(* Logix 5000 project; controller PLC vendor 1 type 14 code 155 rev 32.13; software revision 32.04; part 3 of 5 *)
(* tags used below, declared in another part *)
   Alarm_Word_Current : DINT[3];
   Bridge_Timer_Gearing_Delay : TIMER;
   Bridge_Timer_Gearing_Delay_DN_OS : BOOL;
   Bypass_Encoder : BOOL;   // HMI ENABLE ENCODER
   Depositor : Depositor_R2b;
   FORCE_GO_SIGNAL : BOOL;
   Forces : Forces_R2b;
   homing_timeout : TIMER;
   IO : IO_R2a;
   mv_index_counter : COUNTER;
   MV_indexes : DINT;
   MV_total_indexes : COUNTER;
   NC_NF : NCNF_R2a;   // NC/NF BITSHIFTS
   OS : INT[10];
   Recipe_Setpoints_DINT : DINT[23,20];
   Sequencer_Auto : Sequencer_R2a;
   Sequencer_Home : Sequencer_R2a;
   Servo_MC_Bridge_Shift : Axis_MC_R3b;
   System : System_R2e;
   Timer_Done_Signal_Pulse : TIMER;
   Timers : TIMER[20];   // x
(* MainProgram, continued *)

ROUTINE File_012_Digital_Outputs   (* ladder *)
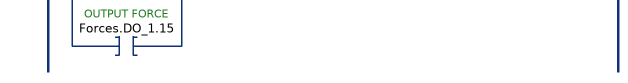
   // DIGITAL OUTPUT MAPPING
   0: [[XIC(IO.DO_1.0) ,XIC(Forces.DO_1.0) ] OTE(Local:1:O.Data.0) ,[XIC(IO.DO_1.1) ,XIC(Forces.DO_1.1) ] OTE(Local:1:O.Data.1) ,[XIC(IO.DO_1.2) ,XIC(Forces.DO_1.2) ] OTE(Local:1:O.Data.2) ,[XIC(IO.DO_1.3) ,XIC(Forces.DO_1.3) ] OTE(Local:1:O.Data.3) ,[XIC(IO.DO_1.4) ,XIC(Forces.DO_1.4) ] OTE(Local:1:O.Data.4) ,[XIC(IO.DO_1.5) ,XIC(Forces.DO_1.5) ] OTE(Local:1:O.Data.5) ,[XIC(IO.DO_1.6) ,XIC(Forces.DO_1.6) ] OTE(Local:1:O.Data.6) ,[XIC(IO.DO_1.7) ,XIC(Forces.DO_1.7) ] OTE(Local:1:O.Data.7) ,[XIC(IO.DO_1.8) ,XIC(Forces.DO_1.8) ] OTE(Local:1:O.Data.8) ,[XIC(IO.DO_1.9) ,XIC(Forces.DO_1.9) ] OTE(Local:1:O.Data.9) ,[XIC(IO.DO_1.10) ,XIC(Forces.DO_1.10) ] OTE(Local:1:O.Data.10) ,[XIC(IO.DO_1.11) ,XIC(Forces.DO_1.11) ] OTE(Local:1:O.Data.11) ,[XIC(IO.DO_1.12) ,XIC(Forces.DO_1.12) ] OTE(Local:1:O.Data.12) ,[XIC(IO.DO_1.13) ,XIC(Forces.DO_1.13) ] OTE(Local:1:O.Data.13) ,[XIC(IO.DO_1.14) ,XIC(Forces.DO_1.14) ] OTE(Local:1:O.Data.14) ,[XIC(IO.DO_1.15) ,XIC(Forces.DO_1.15) ] OTE(Local:1:O.Data.15) ];
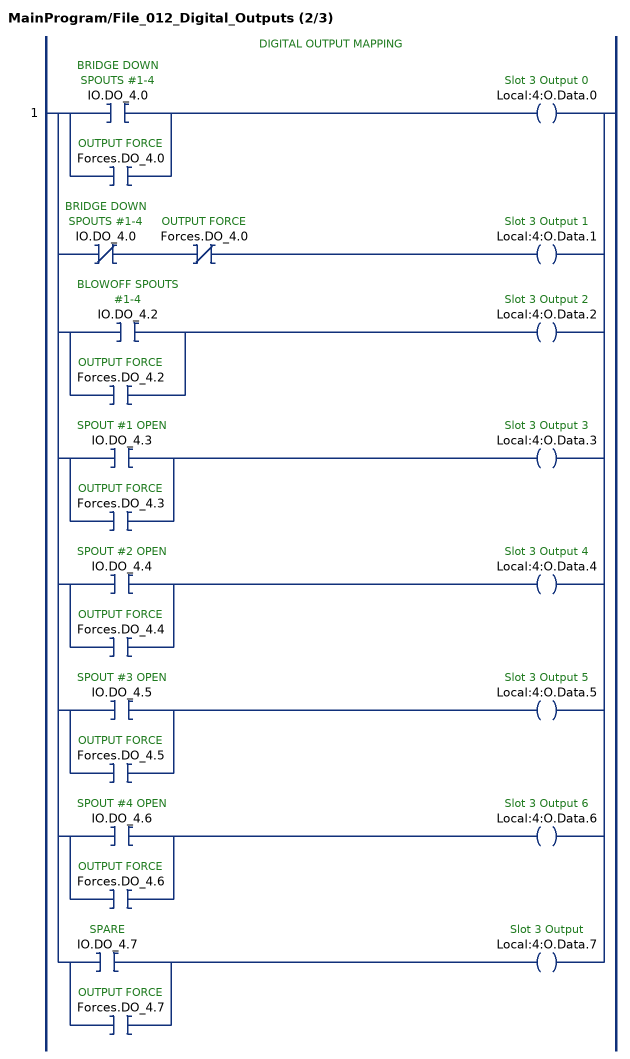
   // DIGITAL OUTPUT MAPPING
   1: [[XIC(IO.DO_4.0) ,XIC(Forces.DO_4.0) ] OTE(Local:4:O.Data.0) ,XIO(IO.DO_4.0) XIO(Forces.DO_4.0) OTE(Local:4:O.Data.1) ,[XIC(IO.DO_4.2) ,XIC(Forces.DO_4.2) ] OTE(Local:4:O.Data.2) ,[XIC(IO.DO_4.3) ,XIC(Forces.DO_4.3) ] OTE(Local:4:O.Data.3) ,[XIC(IO.DO_4.4) ,XIC(Forces.DO_4.4) ] OTE(Local:4:O.Data.4) ,[XIC(IO.DO_4.5) ,XIC(Forces.DO_4.5) ] OTE(Local:4:O.Data.5) ,[XIC(IO.DO_4.6) ,XIC(Forces.DO_4.6) ] OTE(Local:4:O.Data.6) ,[XIC(IO.DO_4.7) ,XIC(Forces.DO_4.7) ] OTE(Local:4:O.Data.7) ];
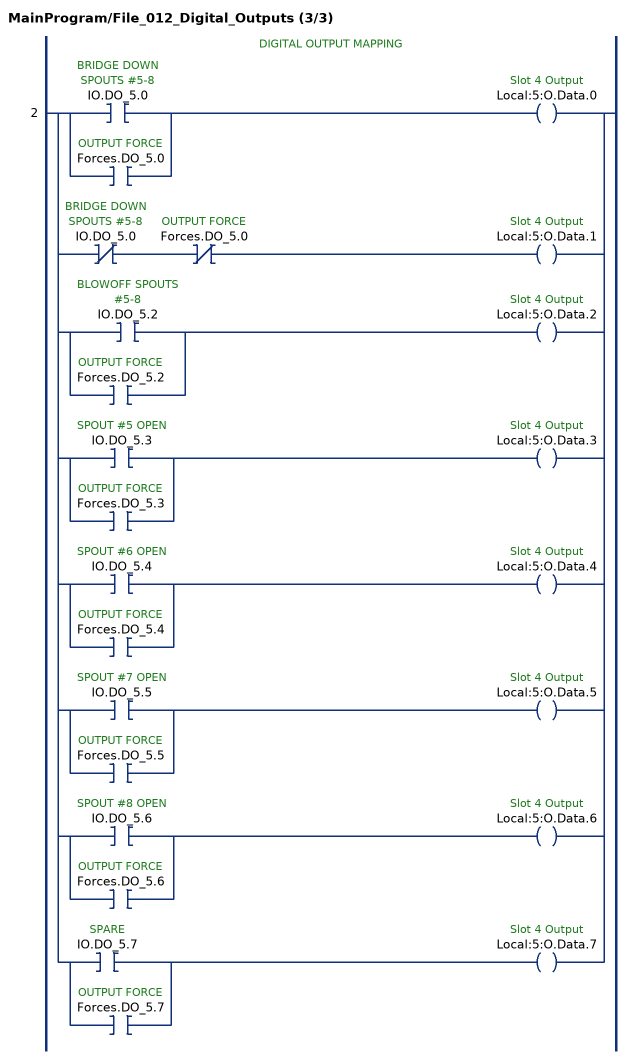
   // DIGITAL OUTPUT MAPPING
   2: [[XIC(IO.DO_5.0) ,XIC(Forces.DO_5.0) ] OTE(Local:5:O.Data.0) ,XIO(IO.DO_5.0) XIO(Forces.DO_5.0) OTE(Local:5:O.Data.1) ,[XIC(IO.DO_5.2) ,XIC(Forces.DO_5.2) ] OTE(Local:5:O.Data.2) ,[XIC(IO.DO_5.3) ,XIC(Forces.DO_5.3) ] OTE(Local:5:O.Data.3) ,[XIC(IO.DO_5.4) ,XIC(Forces.DO_5.4) ] OTE(Local:5:O.Data.4) ,[XIC(IO.DO_5.5) ,XIC(Forces.DO_5.5) ] OTE(Local:5:O.Data.5) ,[XIC(IO.DO_5.6) ,XIC(Forces.DO_5.6) ] OTE(Local:5:O.Data.6) ,[XIC(IO.DO_5.7) ,XIC(Forces.DO_5.7) ] OTE(Local:5:O.Data.7) ];
END_ROUTINE

ROUTINE File_030_Sequencer_Homing   (* ladder *)
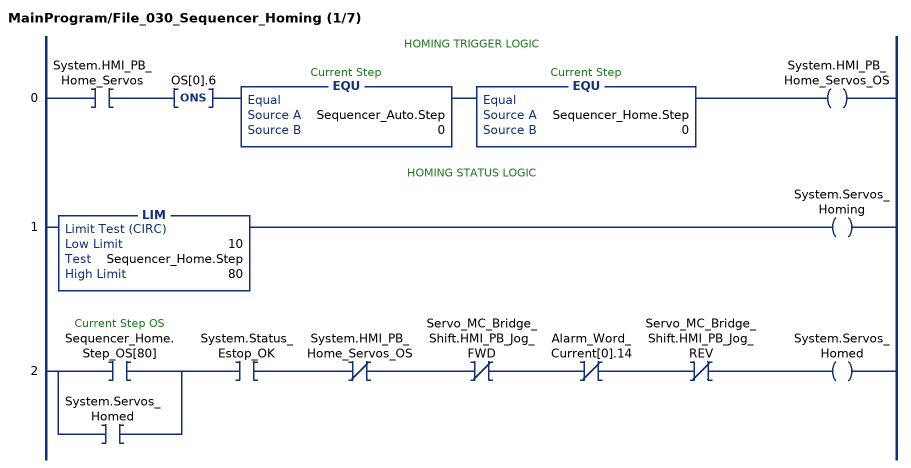
   // HOMING TRIGGER LOGIC
   0: XIC(System.HMI_PB_Home_Servos)ONS(OS[0].6)EQU(Sequencer_Auto.Step,0)EQU(Sequencer_Home.Step,0)OTE(System.HMI_PB_Home_Servos_OS);
   // HOMING STATUS LOGIC
   1: LIM(10,Sequencer_Home.Step,80)OTE(System.Servos_Homing);
   2: [XIC(Sequencer_Home.Step_OS[80]) ,XIC(System.Servos_Homed) ]XIC(System.Status_Estop_OK)XIO(System.HMI_PB_Home_Servos_OS)XIO(Servo_MC_Bridge_Shift.HMI_PB_Jog_FWD)XIO(Alarm_Word_Current[0].14)XIO(Servo_MC_Bridge_Shift.HMI_PB_Jog_REV)OTE(System.Servos_Homed);
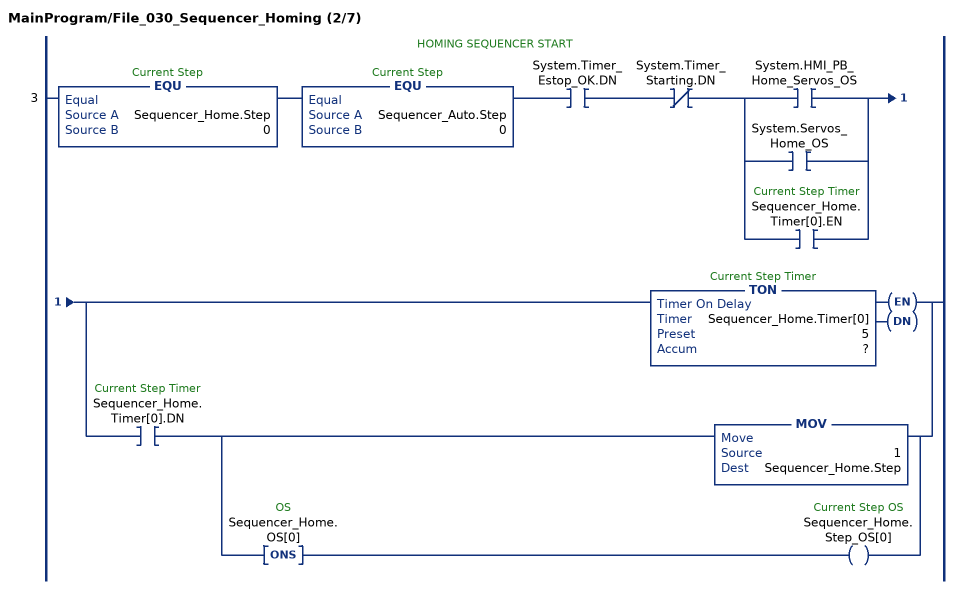
   // HOMING SEQUENCER START
   3: EQU(Sequencer_Home.Step,0)EQU(Sequencer_Auto.Step,0)XIC(System.Timer_Estop_OK.DN)XIO(System.Timer_Starting.DN)[XIC(System.HMI_PB_Home_Servos_OS) ,XIC(System.Servos_Home_OS) ,XIC(Sequencer_Home.Timer[0].EN) ][TON(Sequencer_Home.Timer[0],?,?) ,XIC(Sequencer_Home.Timer[0].DN) [MOV(1,Sequencer_Home.Step) ,ONS(Sequencer_Home.OS[0]) OTE(Sequencer_Home.Step_OS[0]) ] ];
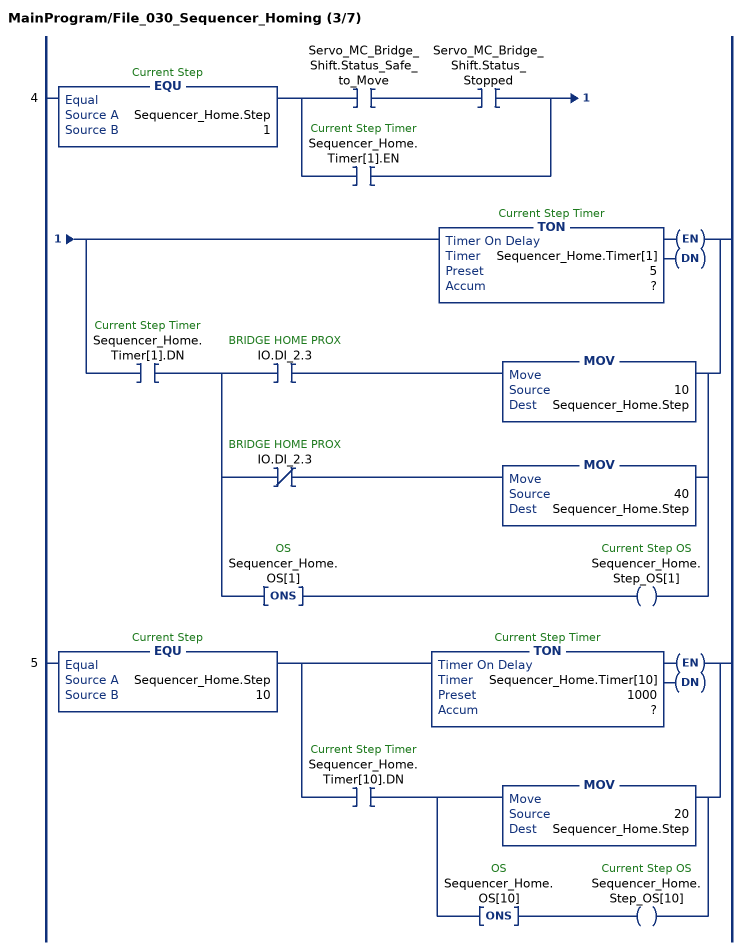
   4: EQU(Sequencer_Home.Step,1)[XIC(Servo_MC_Bridge_Shift.Status_Safe_to_Move) XIC(Servo_MC_Bridge_Shift.Status_Stopped) ,XIC(Sequencer_Home.Timer[1].EN) ][TON(Sequencer_Home.Timer[1],?,?) ,XIC(Sequencer_Home.Timer[1].DN) [XIC(IO.DI_2.3) MOV(10,Sequencer_Home.Step) ,XIO(IO.DI_2.3) MOV(40,Sequencer_Home.Step) ,ONS(Sequencer_Home.OS[1]) OTE(Sequencer_Home.Step_OS[1]) ] ];
   5: EQU(Sequencer_Home.Step,10)[TON(Sequencer_Home.Timer[10],?,?) ,XIC(Sequencer_Home.Timer[10].DN) [MOV(20,Sequencer_Home.Step) ,ONS(Sequencer_Home.OS[10]) OTE(Sequencer_Home.Step_OS[10]) ] ];
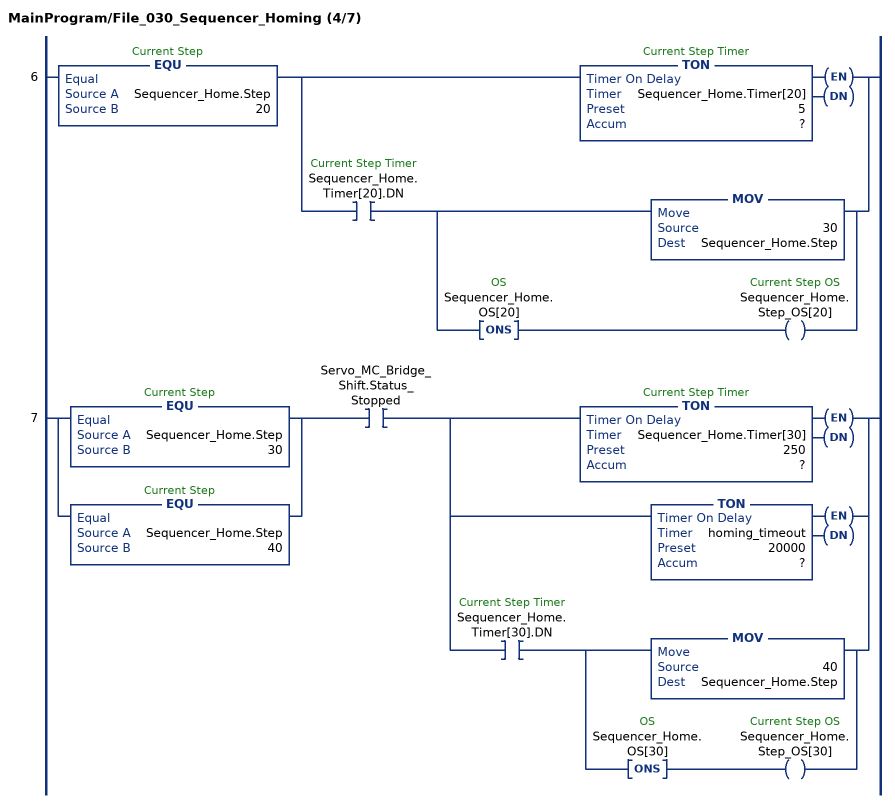
   6: EQU(Sequencer_Home.Step,20)[TON(Sequencer_Home.Timer[20],?,?) ,XIC(Sequencer_Home.Timer[20].DN) [MOV(30,Sequencer_Home.Step) ,ONS(Sequencer_Home.OS[20]) OTE(Sequencer_Home.Step_OS[20]) ] ];
   7: [EQU(Sequencer_Home.Step,30) ,EQU(Sequencer_Home.Step,40) ]XIC(Servo_MC_Bridge_Shift.Status_Stopped)[[TON(Sequencer_Home.Timer[30],?,?) ,TON(homing_timeout,?,?) ] ,XIC(Sequencer_Home.Timer[30].DN) [MOV(40,Sequencer_Home.Step) ,ONS(Sequencer_Home.OS[30]) OTE(Sequencer_Home.Step_OS[30]) ] ];
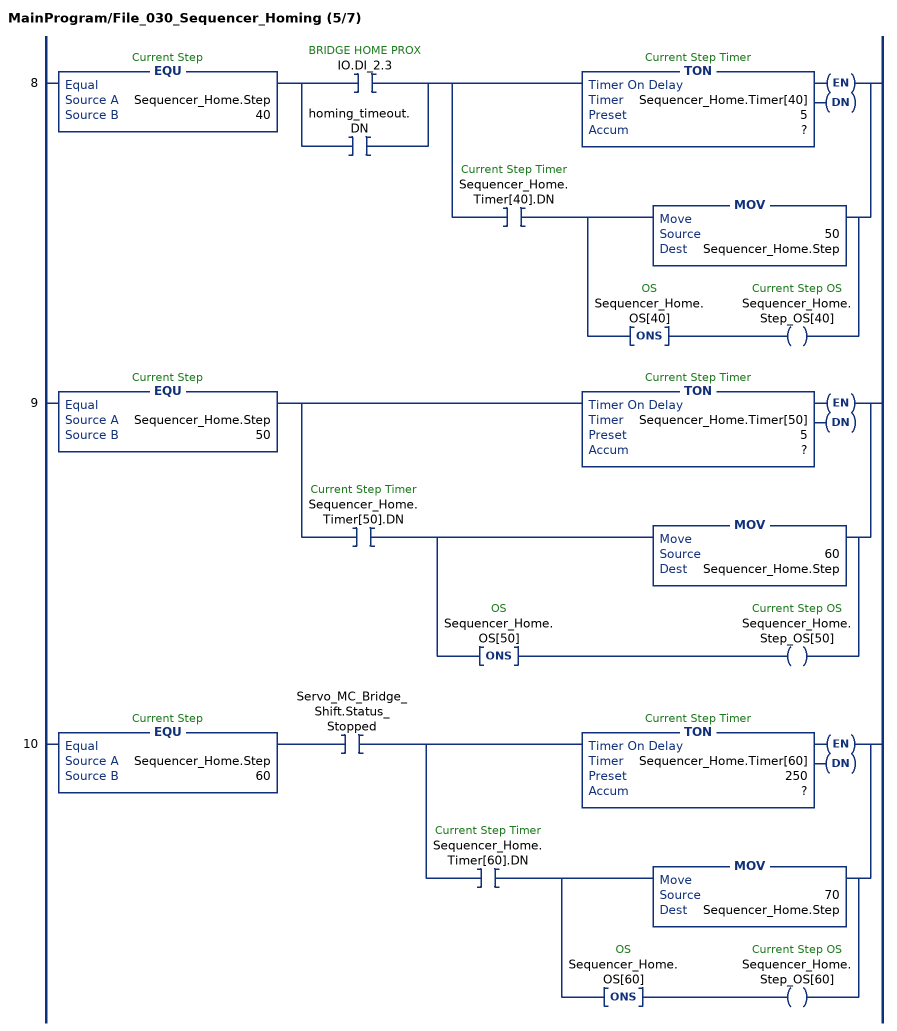
   8: EQU(Sequencer_Home.Step,40)[XIC(IO.DI_2.3) ,XIC(homing_timeout.DN) ][TON(Sequencer_Home.Timer[40],?,?) ,XIC(Sequencer_Home.Timer[40].DN) [MOV(50,Sequencer_Home.Step) ,ONS(Sequencer_Home.OS[40]) OTE(Sequencer_Home.Step_OS[40]) ] ];
   9: EQU(Sequencer_Home.Step,50)[TON(Sequencer_Home.Timer[50],?,?) ,XIC(Sequencer_Home.Timer[50].DN) [MOV(60,Sequencer_Home.Step) ,ONS(Sequencer_Home.OS[50]) OTE(Sequencer_Home.Step_OS[50]) ] ];
   10: EQU(Sequencer_Home.Step,60)XIC(Servo_MC_Bridge_Shift.Status_Stopped)[TON(Sequencer_Home.Timer[60],?,?) ,XIC(Sequencer_Home.Timer[60].DN) [MOV(70,Sequencer_Home.Step) ,ONS(Sequencer_Home.OS[60]) OTE(Sequencer_Home.Step_OS[60]) ] ];
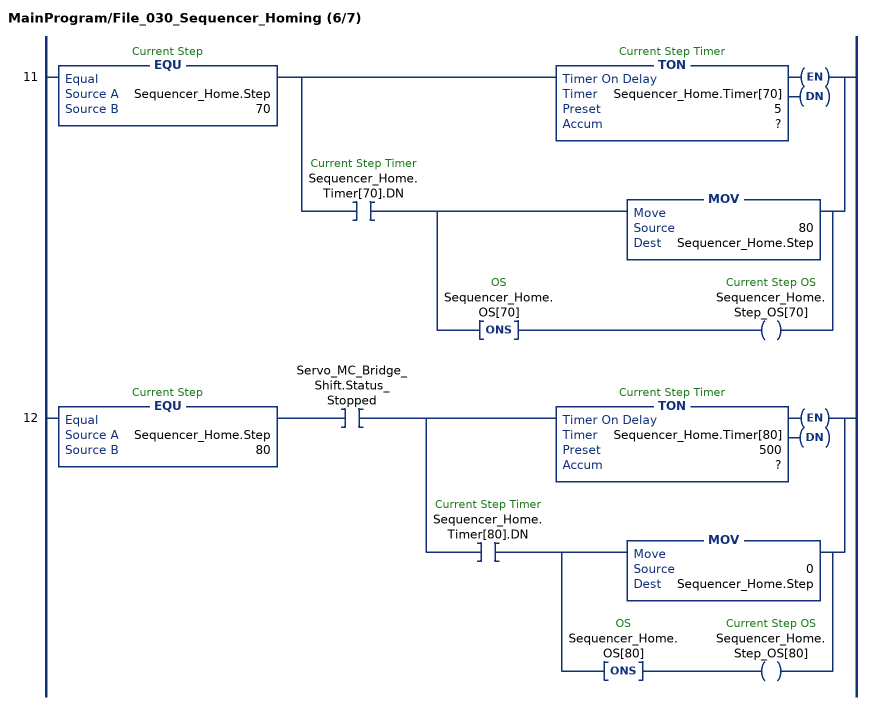
   11: EQU(Sequencer_Home.Step,70)[TON(Sequencer_Home.Timer[70],?,?) ,XIC(Sequencer_Home.Timer[70].DN) [MOV(80,Sequencer_Home.Step) ,ONS(Sequencer_Home.OS[70]) OTE(Sequencer_Home.Step_OS[70]) ] ];
   12: EQU(Sequencer_Home.Step,80)XIC(Servo_MC_Bridge_Shift.Status_Stopped)[TON(Sequencer_Home.Timer[80],?,?) ,XIC(Sequencer_Home.Timer[80].DN) [MOV(0,Sequencer_Home.Step) ,ONS(Sequencer_Home.OS[80]) OTE(Sequencer_Home.Step_OS[80]) ] ];
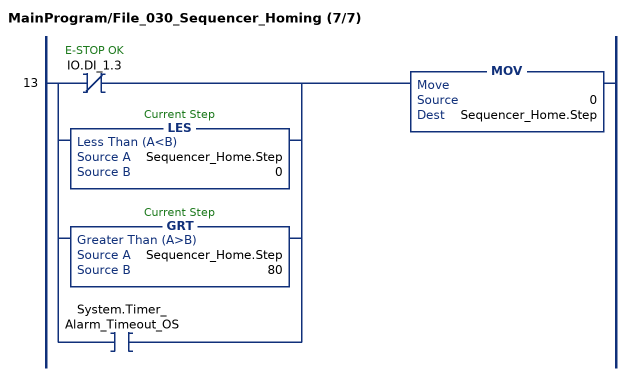
   13: [XIO(IO.DI_1.3) ,LES(Sequencer_Home.Step,0) ,GRT(Sequencer_Home.Step,80) ,XIC(System.Timer_Alarm_Timeout_OS) ]MOV(0,Sequencer_Home.Step);
END_ROUTINE

ROUTINE File_040_Sequencer_Auto   (* ladder *)
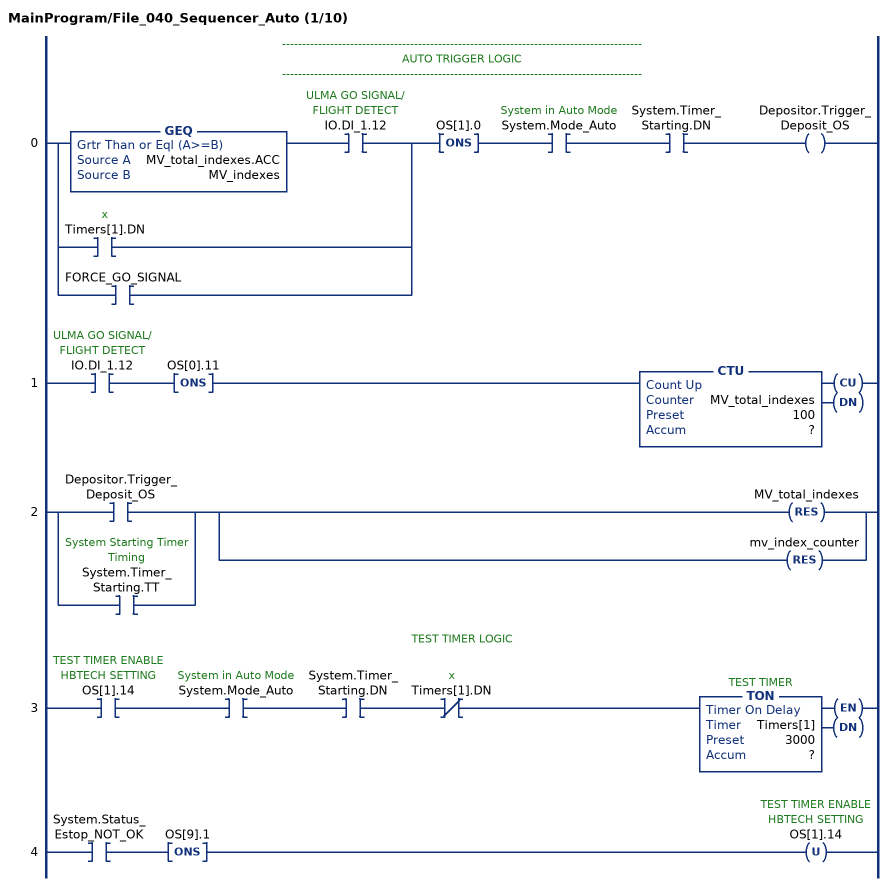
   // ------------------------------------------------------------------------------------------
   // AUTO TRIGGER LOGIC
   // ------------------------------------------------------------------------------------------
   0: [GEQ(MV_total_indexes.ACC,MV_indexes) XIC(IO.DI_1.12) ,XIC(Timers[1].DN) ,XIC(FORCE_GO_SIGNAL) ]ONS(OS[1].0)XIC(System.Mode_Auto)XIC(System.Timer_Starting.DN)OTE(Depositor.Trigger_Deposit_OS);
   1: XIC(IO.DI_1.12)ONS(OS[0].11)CTU(MV_total_indexes,?,?);
   2: [XIC(Depositor.Trigger_Deposit_OS) ,XIC(System.Timer_Starting.TT) ][RES(MV_total_indexes) ,RES(mv_index_counter) ];
   // TEST TIMER LOGIC
   3: XIC(OS[1].14)XIC(System.Mode_Auto)XIC(System.Timer_Starting.DN)XIO(Timers[1].DN)TON(Timers[1],?,?);
   4: XIC(System.Status_Estop_NOT_OK)ONS(OS[9].1)OTU(OS[1].14);
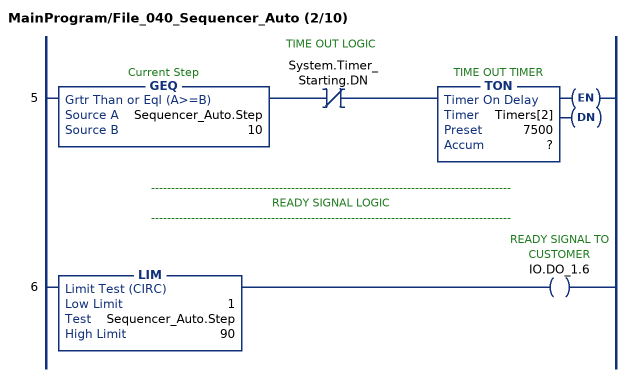
   // TIME OUT LOGIC
   5: GEQ(Sequencer_Auto.Step,10)XIO(System.Timer_Starting.DN)TON(Timers[2],?,?);
   // ------------------------------------------------------------------------------------------
   // READY SIGNAL LOGIC
   // ------------------------------------------------------------------------------------------
   6: LIM(1,Sequencer_Auto.Step,90)OTE(IO.DO_1.6);
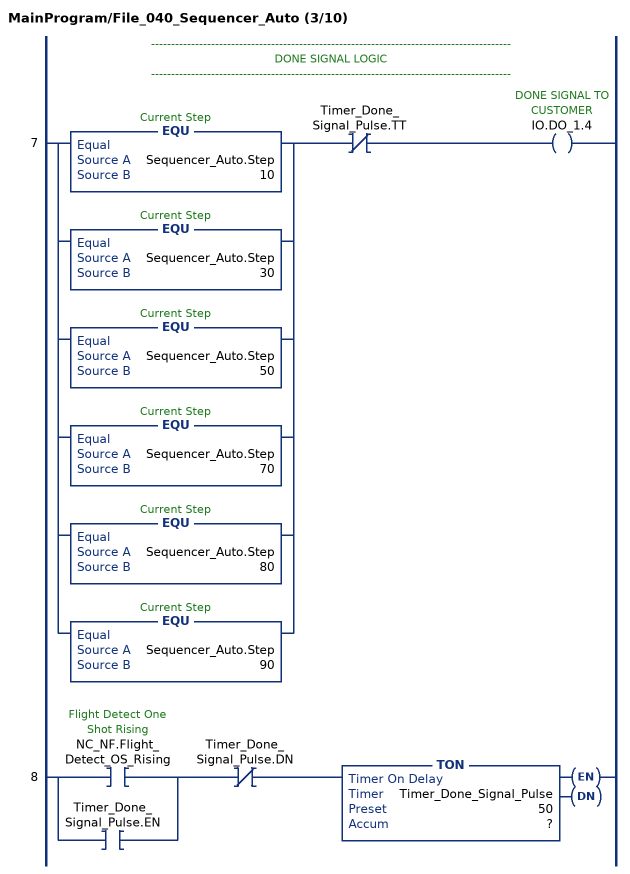
   // ------------------------------------------------------------------------------------------
   // DONE SIGNAL LOGIC
   // ------------------------------------------------------------------------------------------
   7: [EQU(Sequencer_Auto.Step,10) ,EQU(Sequencer_Auto.Step,30) ,EQU(Sequencer_Auto.Step,50) ,EQU(Sequencer_Auto.Step,70) ,EQU(Sequencer_Auto.Step,80) ,EQU(Sequencer_Auto.Step,90) ]XIO(Timer_Done_Signal_Pulse.TT)OTE(IO.DO_1.4);
   8: [XIC(NC_NF.Flight_Detect_OS_Rising) ,XIC(Timer_Done_Signal_Pulse.EN) ]XIO(Timer_Done_Signal_Pulse.DN)TON(Timer_Done_Signal_Pulse,?,?);
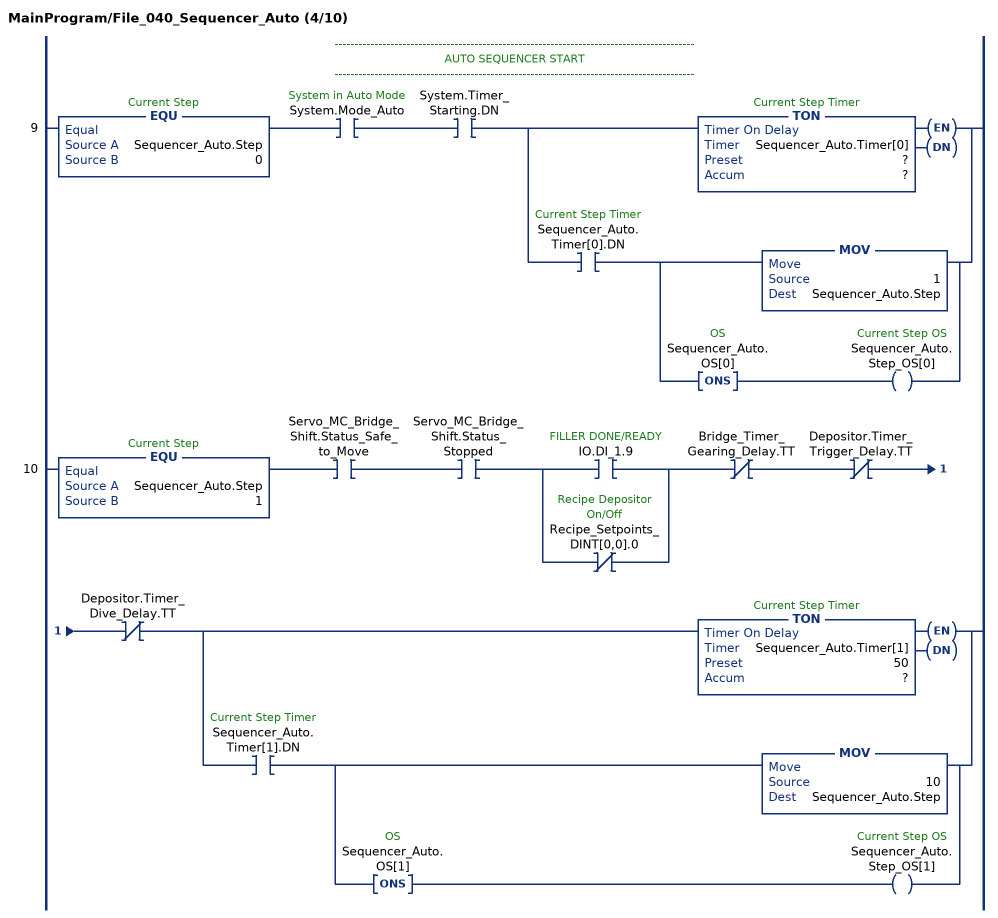
   // ------------------------------------------------------------------------------------------
   // AUTO SEQUENCER START
   // ------------------------------------------------------------------------------------------
   9: EQU(Sequencer_Auto.Step,0)XIC(System.Mode_Auto)XIC(System.Timer_Starting.DN)[TON(Sequencer_Auto.Timer[0],?,?) ,XIC(Sequencer_Auto.Timer[0].DN) [MOV(1,Sequencer_Auto.Step) ,ONS(Sequencer_Auto.OS[0]) OTE(Sequencer_Auto.Step_OS[0]) ] ];
   10: EQU(Sequencer_Auto.Step,1)XIC(Servo_MC_Bridge_Shift.Status_Safe_to_Move)XIC(Servo_MC_Bridge_Shift.Status_Stopped)[XIC(IO.DI_1.9) ,XIO(Recipe_Setpoints_DINT[0,0].0) ]XIO(Bridge_Timer_Gearing_Delay.TT)XIO(Depositor.Timer_Trigger_Delay.TT)XIO(Depositor.Timer_Dive_Delay.TT)[TON(Sequencer_Auto.Timer[1],?,?) ,XIC(Sequencer_Auto.Timer[1].DN) [MOV(10,Sequencer_Auto.Step) ,ONS(Sequencer_Auto.OS[1]) OTE(Sequencer_Auto.Step_OS[1]) ] ];
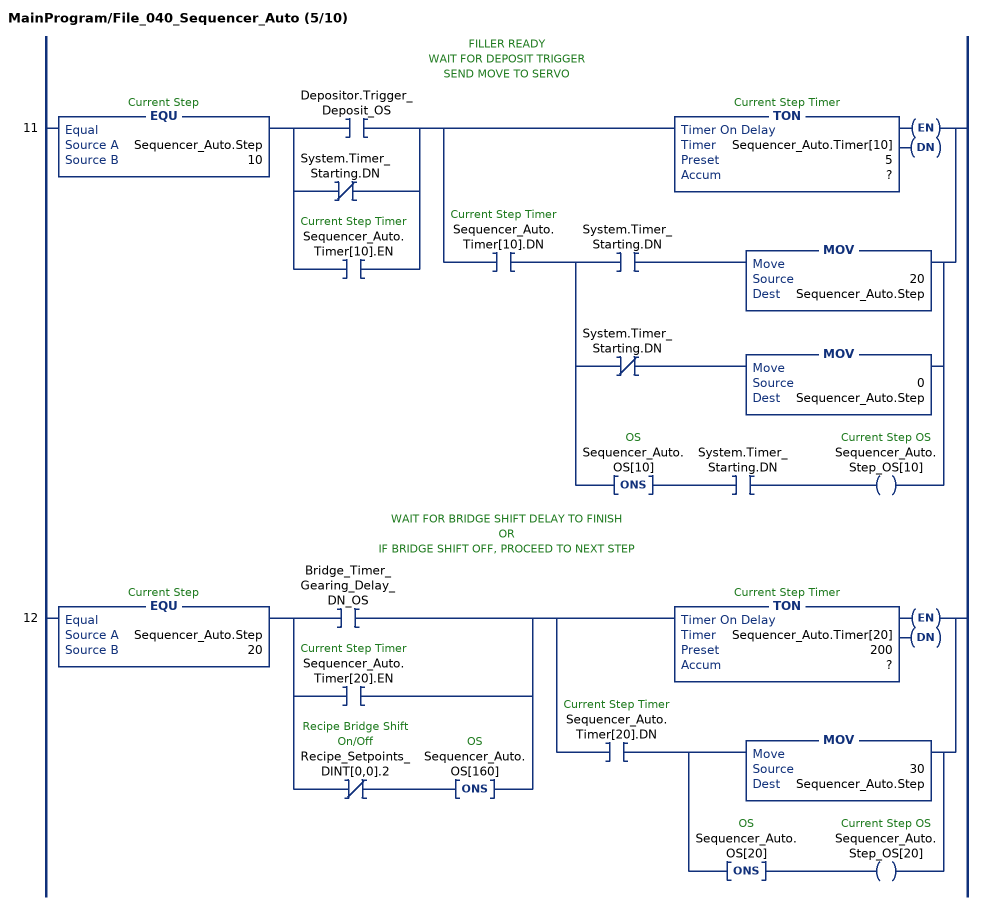
   // FILLER READY
   // WAIT FOR DEPOSIT TRIGGER
   // SEND MOVE TO SERVO
   11: EQU(Sequencer_Auto.Step,10)[XIC(Depositor.Trigger_Deposit_OS) ,XIO(System.Timer_Starting.DN) ,XIC(Sequencer_Auto.Timer[10].EN) ][TON(Sequencer_Auto.Timer[10],?,?) ,XIC(Sequencer_Auto.Timer[10].DN) [XIC(System.Timer_Starting.DN) MOV(20,Sequencer_Auto.Step) ,XIO(System.Timer_Starting.DN) MOV(0,Sequencer_Auto.Step) ,ONS(Sequencer_Auto.OS[10]) XIC(System.Timer_Starting.DN) OTE(Sequencer_Auto.Step_OS[10]) ] ];
   // WAIT FOR BRIDGE SHIFT DELAY TO FINISH
   // OR
   // IF BRIDGE SHIFT OFF, PROCEED TO NEXT STEP
   12: EQU(Sequencer_Auto.Step,20)[XIC(Bridge_Timer_Gearing_Delay_DN_OS) ,XIC(Sequencer_Auto.Timer[20].EN) ,XIO(Recipe_Setpoints_DINT[0,0].2) ONS(Sequencer_Auto.OS[160]) ][TON(Sequencer_Auto.Timer[20],?,?) ,XIC(Sequencer_Auto.Timer[20].DN) [MOV(30,Sequencer_Auto.Step) ,ONS(Sequencer_Auto.OS[20]) OTE(Sequencer_Auto.Step_OS[20]) ] ];
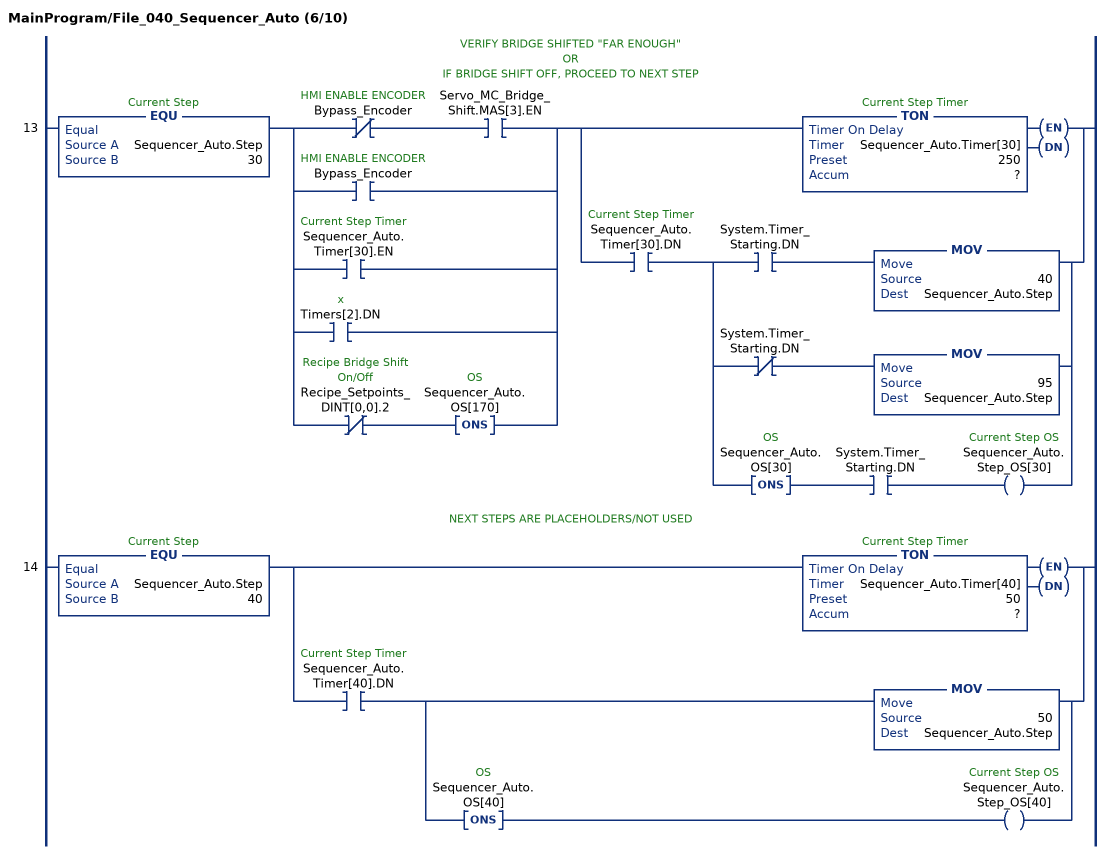
   // VERIFY BRIDGE SHIFTED "FAR ENOUGH"
   // OR
   // IF BRIDGE SHIFT OFF, PROCEED TO NEXT STEP
   13: EQU(Sequencer_Auto.Step,30)[XIO(Bypass_Encoder) XIC(Servo_MC_Bridge_Shift.MAS[3].EN) ,XIC(Bypass_Encoder) ,XIC(Sequencer_Auto.Timer[30].EN) ,XIC(Timers[2].DN) ,XIO(Recipe_Setpoints_DINT[0,0].2) ONS(Sequencer_Auto.OS[170]) ][TON(Sequencer_Auto.Timer[30],?,?) ,XIC(Sequencer_Auto.Timer[30].DN) [XIC(System.Timer_Starting.DN) MOV(40,Sequencer_Auto.Step) ,XIO(System.Timer_Starting.DN) MOV(95,Sequencer_Auto.Step) ,ONS(Sequencer_Auto.OS[30]) XIC(System.Timer_Starting.DN) OTE(Sequencer_Auto.Step_OS[30]) ] ];
   // NEXT STEPS ARE PLACEHOLDERS/NOT USED
   14: EQU(Sequencer_Auto.Step,40)[TON(Sequencer_Auto.Timer[40],?,?) ,XIC(Sequencer_Auto.Timer[40].DN) [MOV(50,Sequencer_Auto.Step) ,ONS(Sequencer_Auto.OS[40]) OTE(Sequencer_Auto.Step_OS[40]) ] ];
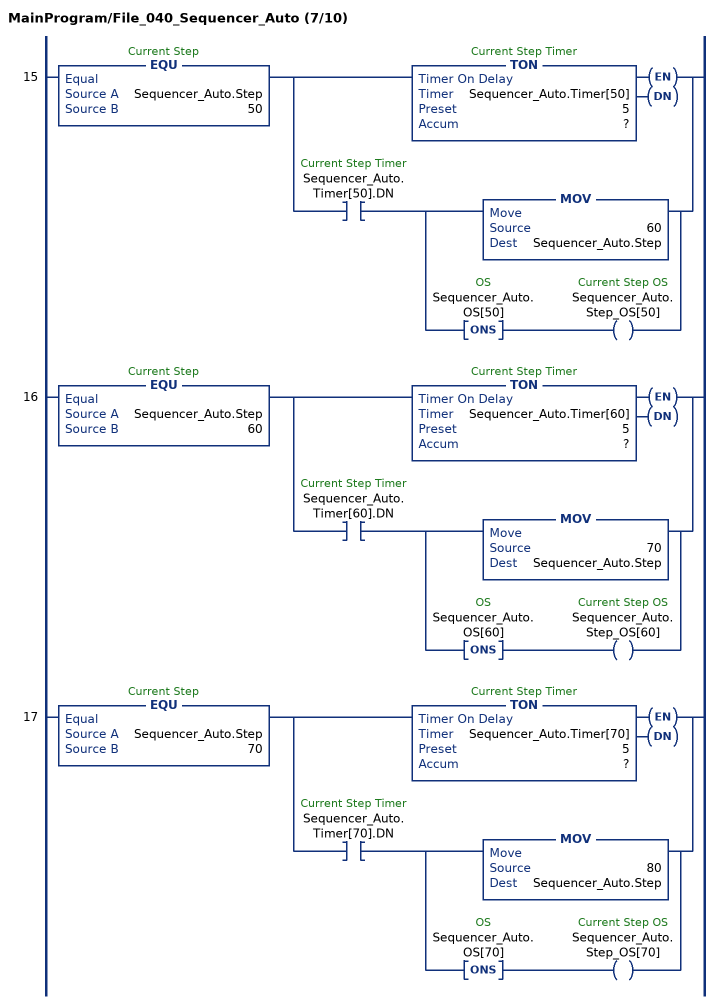
   15: EQU(Sequencer_Auto.Step,50)[TON(Sequencer_Auto.Timer[50],?,?) ,XIC(Sequencer_Auto.Timer[50].DN) [MOV(60,Sequencer_Auto.Step) ,ONS(Sequencer_Auto.OS[50]) OTE(Sequencer_Auto.Step_OS[50]) ] ];
   16: EQU(Sequencer_Auto.Step,60)[TON(Sequencer_Auto.Timer[60],?,?) ,XIC(Sequencer_Auto.Timer[60].DN) [MOV(70,Sequencer_Auto.Step) ,ONS(Sequencer_Auto.OS[60]) OTE(Sequencer_Auto.Step_OS[60]) ] ];
   17: EQU(Sequencer_Auto.Step,70)[TON(Sequencer_Auto.Timer[70],?,?) ,XIC(Sequencer_Auto.Timer[70].DN) [MOV(80,Sequencer_Auto.Step) ,ONS(Sequencer_Auto.OS[70]) OTE(Sequencer_Auto.Step_OS[70]) ] ];
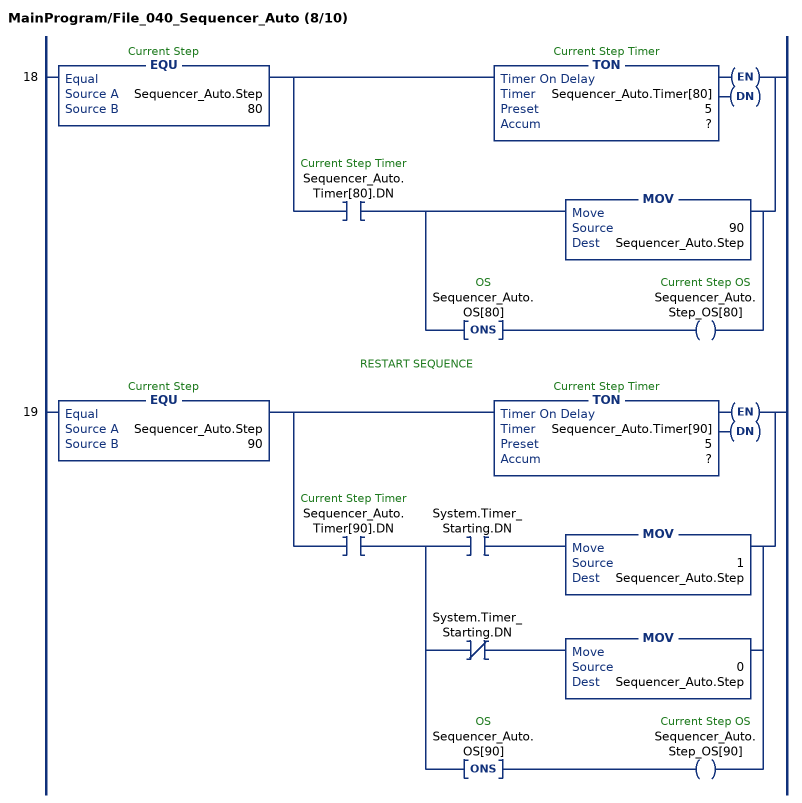
   18: EQU(Sequencer_Auto.Step,80)[TON(Sequencer_Auto.Timer[80],?,?) ,XIC(Sequencer_Auto.Timer[80].DN) [MOV(90,Sequencer_Auto.Step) ,ONS(Sequencer_Auto.OS[80]) OTE(Sequencer_Auto.Step_OS[80]) ] ];
   // RESTART SEQUENCE
   19: EQU(Sequencer_Auto.Step,90)[TON(Sequencer_Auto.Timer[90],?,?) ,XIC(Sequencer_Auto.Timer[90].DN) [XIC(System.Timer_Starting.DN) MOV(1,Sequencer_Auto.Step) ,XIO(System.Timer_Starting.DN) MOV(0,Sequencer_Auto.Step) ,ONS(Sequencer_Auto.OS[90]) OTE(Sequencer_Auto.Step_OS[90]) ] ];
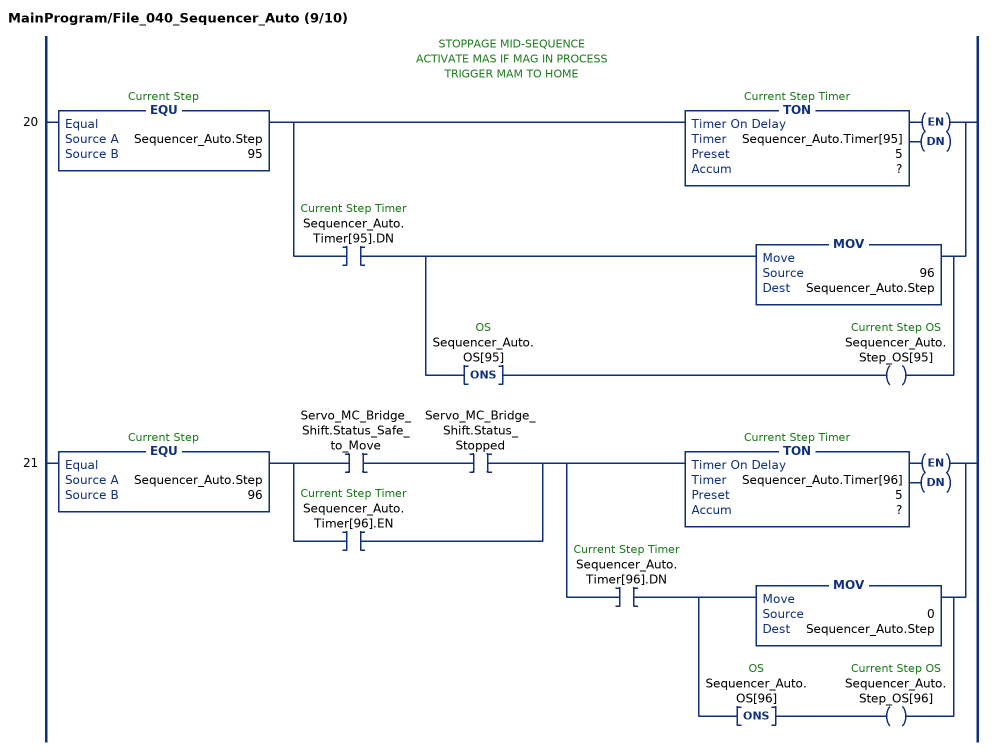
   // STOPPAGE MID-SEQUENCE
   // ACTIVATE MAS IF MAG IN PROCESS
   // TRIGGER MAM TO HOME
   20: EQU(Sequencer_Auto.Step,95)[TON(Sequencer_Auto.Timer[95],?,?) ,XIC(Sequencer_Auto.Timer[95].DN) [MOV(96,Sequencer_Auto.Step) ,ONS(Sequencer_Auto.OS[95]) OTE(Sequencer_Auto.Step_OS[95]) ] ];
   21: EQU(Sequencer_Auto.Step,96)[XIC(Servo_MC_Bridge_Shift.Status_Safe_to_Move) XIC(Servo_MC_Bridge_Shift.Status_Stopped) ,XIC(Sequencer_Auto.Timer[96].EN) ][TON(Sequencer_Auto.Timer[96],?,?) ,XIC(Sequencer_Auto.Timer[96].DN) [MOV(0,Sequencer_Auto.Step) ,ONS(Sequencer_Auto.OS[96]) OTE(Sequencer_Auto.Step_OS[96]) ] ];
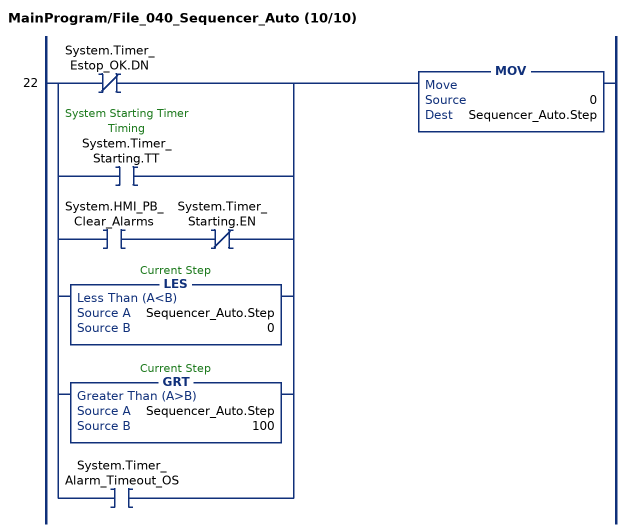
   22: [XIO(System.Timer_Estop_OK.DN) ,XIC(System.Timer_Starting.TT) ,XIC(System.HMI_PB_Clear_Alarms) XIO(System.Timer_Starting.EN) ,LES(Sequencer_Auto.Step,0) ,GRT(Sequencer_Auto.Step,100) ,XIC(System.Timer_Alarm_Timeout_OS) ]MOV(0,Sequencer_Auto.Step);
END_ROUTINE
